{attribute addProperty BoxType "EK1122-0000-0018"}
{attribute addProperty Id "Beckhoff_EP3xxxsub_EK1100EK1100_179A0949162A_0001_EP3162_0002_0016EP3162_C6F348DD14618.25A_0002_EP3162_1002_0017EP3162_F6B2922016220.25A_0003_EP3174_0002_0016EP3174_360D511E40650.75A_0004_EP3174_0002_0017EP3174_360D511E40650.75A_0005_EP3174_0002_0018EP3174_6082EBFD21026.25A_0006_EP3174_0002_0019EP3174_6082EBFD21026.25A_0007_EP3174_0002_0020EP3174_B7B5302521026.25A_0008_EP3174_0002_0021EP3174_B7B5302521026.25A_0009_EP3174_0002_0022EP3174_B7B5302521026.25A_0010_EP3174_0002_0023EP3174_B7B5302521026.25A_0011_EP3174_0092_0016EP3174_B7B5302521026.25A_0012_EP3182_1002_0017EP3182_12747D8E16220.25A_0013_EP3182_1002_0018EP3182_F6B2922016220.25A_0014_EP3182_1002_0019EP3182_F6B2922016220.25A_0015_EP3182_1002_0020EP3182_F6B2922016220.25A_0016_EP3184_0002_0016EP3184_360D511E40650.75A_0017_EP3184_0002_0017EP3184_6082EBFD21026.25A_0018_EP3184_0002_0018EP3184_6082EBFD21026.25A_0019_EP3184_0002_0019EP3184_6082EBFD21026.25A_0020_EP3184_0002_0020EP3184_6082EBFD21026.25A_0021_EP3184_0002_0021EP3184_B7B5302521026.25A_0022_EP3184_0402_0016EP3184_6082EBFD21026.25A_0023_EP3184_0402_0017EP3184_6082EBFD21026.25A_0024_EP3184_0402_0018EP3184_B7B5302521026.25A_0025_EP3184_1002_0016EP3184_360D511E40650.75A_0026_EP3184_1002_0017EP3184_360D511E40650.75A_0027_EP3184_1002_0018EP3184_6082EBFD21026.25A_0028_EP3184_1002_0019EP3184_6082EBFD21026.25A_0029_EP3184_1002_0020EP3184_6082EBFD21026.25A_0030_EP3184_1002_0021EP3184_B7B5302521026.25A_0031_EP3204_0002_0017EP3204_72ABB95437847.25A_0032_EP3204_0002_0018EP3204_72ABB95437847.25A_0033_EP3204_0002_0019EP3204_72ABB95437847.25A_0034_EP3204_0002_0020EP3204_72ABB95437847.25A_0035_EP3204_0002_0021EP3204_C91659E221026.25A_0036_EP3314_0002_0016EP3314_3064F86237847.25A_0037_EP3314_0002_0017EP3314_3064F86237847.25A_0038_EP3314_0002_0018EP3314_1D3C92AC21026.25A_0039_EP3314_0002_0019EP3314_A69716D721026.25A_0040_EP3314_0002_0020EP3314_A69716D721026.25A_0041_EP3314_0002_0021EP3314_A69716D721026.25A_0042_EP3351_2022_0016EP3351_952A9D2322628.25A_0043_EP3356_0022_0016EP3356_AAE78EE214618.25A_0044_EP3356_0022_0017EP3356_AAE78EE214618.25A_0045_EP3356_0022_0022EP3356_AAE78EE214618.25A_0046_EP3632_0001_0016EP3632_A724E07457872.25A_0047_EP3632_0001_0017EP3632_A724E07457872.25A_0048_EP3744_0041_0016EP3744_99A8040A38648.25A_0049_EP3744_0041_0017EP3744_99A8040A38648.25A_0050_EP3744_0041_0018EP3744_99A8040A38648.25A_0051_EP3744_0041_0019EP3744_99A8040A38648.25A_0052_EP3744_0041_0020EP3744_99A8040A38648.25A_0053_EP3744_0041_0021EP3744_99A8040A38648.25A_0054_EP3744_1041_0016EP3744_99A8040A38648.25A_0055_EP3744_1041_0017EP3744_99A8040A38648.25A_0056_EP3744_1041_0018EP3744_99A8040A38648.25A_0057_EP3744_1041_0019EP3744_99A8040A38648.25A_0058_EP3744_1041_0020EP3744_99A8040A38648.25A_0059_EP3744_1041_0021EP3744_99A8040A38648.25A_0060_EP3752_0000_0017EP3752_639ED5F327434.25A_0061_EP3752_0000_0018EP3752_639ED5F327434.25"}
{attribute addProperty CRC "2518642837"}
{attribute addProperty SizeInBites "17310"}
{attribute addProperty SizeInBytes "2163.75"}
TYPE Beckhoff_EP3xxxEK1122_961F7095 EXTENDS EK1122_179A0949 :
STRUCT
	{attribute addProperty Name "Beckhoff_EP3xxxsub_EK1100"}
	Beckhoff_EP3xxxsub_EK1100 : EK1100_179A0949;
	{attribute addProperty Name "A_0001_EP3162_0002_0016"}
	A_0001_EP3162_0002_0016 : EP3162_C6F348DD;
	{attribute addProperty Name "A_0002_EP3162_1002_0017"}
	A_0002_EP3162_1002_0017 : EP3162_F6B29220;
	{attribute addProperty Name "A_0003_EP3174_0002_0016"}
	A_0003_EP3174_0002_0016 : EP3174_360D511E;
	{attribute addProperty Name "A_0004_EP3174_0002_0017"}
	A_0004_EP3174_0002_0017 : EP3174_360D511E;
	{attribute addProperty Name "A_0005_EP3174_0002_0018"}
	A_0005_EP3174_0002_0018 : EP3174_6082EBFD;
	{attribute addProperty Name "A_0006_EP3174_0002_0019"}
	A_0006_EP3174_0002_0019 : EP3174_6082EBFD;
	{attribute addProperty Name "A_0007_EP3174_0002_0020"}
	A_0007_EP3174_0002_0020 : EP3174_B7B53025;
	{attribute addProperty Name "A_0008_EP3174_0002_0021"}
	A_0008_EP3174_0002_0021 : EP3174_B7B53025;
	{attribute addProperty Name "A_0009_EP3174_0002_0022"}
	A_0009_EP3174_0002_0022 : EP3174_B7B53025;
	{attribute addProperty Name "A_0010_EP3174_0002_0023"}
	A_0010_EP3174_0002_0023 : EP3174_B7B53025;
	{attribute addProperty Name "A_0011_EP3174_0092_0016"}
	A_0011_EP3174_0092_0016 : EP3174_B7B53025;
	{attribute addProperty Name "A_0012_EP3182_1002_0017"}
	A_0012_EP3182_1002_0017 : EP3182_12747D8E;
	{attribute addProperty Name "A_0013_EP3182_1002_0018"}
	A_0013_EP3182_1002_0018 : EP3182_F6B29220;
	{attribute addProperty Name "A_0014_EP3182_1002_0019"}
	A_0014_EP3182_1002_0019 : EP3182_F6B29220;
	{attribute addProperty Name "A_0015_EP3182_1002_0020"}
	A_0015_EP3182_1002_0020 : EP3182_F6B29220;
	{attribute addProperty Name "A_0016_EP3184_0002_0016"}
	A_0016_EP3184_0002_0016 : EP3184_360D511E;
	{attribute addProperty Name "A_0017_EP3184_0002_0017"}
	A_0017_EP3184_0002_0017 : EP3184_6082EBFD;
	{attribute addProperty Name "A_0018_EP3184_0002_0018"}
	A_0018_EP3184_0002_0018 : EP3184_6082EBFD;
	{attribute addProperty Name "A_0019_EP3184_0002_0019"}
	A_0019_EP3184_0002_0019 : EP3184_6082EBFD;
	{attribute addProperty Name "A_0020_EP3184_0002_0020"}
	A_0020_EP3184_0002_0020 : EP3184_6082EBFD;
	{attribute addProperty Name "A_0021_EP3184_0002_0021"}
	A_0021_EP3184_0002_0021 : EP3184_B7B53025;
	{attribute addProperty Name "A_0022_EP3184_0402_0016"}
	A_0022_EP3184_0402_0016 : EP3184_6082EBFD;
	{attribute addProperty Name "A_0023_EP3184_0402_0017"}
	A_0023_EP3184_0402_0017 : EP3184_6082EBFD;
	{attribute addProperty Name "A_0024_EP3184_0402_0018"}
	A_0024_EP3184_0402_0018 : EP3184_B7B53025;
	{attribute addProperty Name "A_0025_EP3184_1002_0016"}
	A_0025_EP3184_1002_0016 : EP3184_360D511E;
	{attribute addProperty Name "A_0026_EP3184_1002_0017"}
	A_0026_EP3184_1002_0017 : EP3184_360D511E;
	{attribute addProperty Name "A_0027_EP3184_1002_0018"}
	A_0027_EP3184_1002_0018 : EP3184_6082EBFD;
	{attribute addProperty Name "A_0028_EP3184_1002_0019"}
	A_0028_EP3184_1002_0019 : EP3184_6082EBFD;
	{attribute addProperty Name "A_0029_EP3184_1002_0020"}
	A_0029_EP3184_1002_0020 : EP3184_6082EBFD;
	{attribute addProperty Name "A_0030_EP3184_1002_0021"}
	A_0030_EP3184_1002_0021 : EP3184_B7B53025;
	{attribute addProperty Name "A_0031_EP3204_0002_0017"}
	A_0031_EP3204_0002_0017 : EP3204_72ABB954;
	{attribute addProperty Name "A_0032_EP3204_0002_0018"}
	A_0032_EP3204_0002_0018 : EP3204_72ABB954;
	{attribute addProperty Name "A_0033_EP3204_0002_0019"}
	A_0033_EP3204_0002_0019 : EP3204_72ABB954;
	{attribute addProperty Name "A_0034_EP3204_0002_0020"}
	A_0034_EP3204_0002_0020 : EP3204_72ABB954;
	{attribute addProperty Name "A_0035_EP3204_0002_0021"}
	A_0035_EP3204_0002_0021 : EP3204_C91659E2;
	{attribute addProperty Name "A_0036_EP3314_0002_0016"}
	A_0036_EP3314_0002_0016 : EP3314_3064F862;
	{attribute addProperty Name "A_0037_EP3314_0002_0017"}
	A_0037_EP3314_0002_0017 : EP3314_3064F862;
	{attribute addProperty Name "A_0038_EP3314_0002_0018"}
	A_0038_EP3314_0002_0018 : EP3314_1D3C92AC;
	{attribute addProperty Name "A_0039_EP3314_0002_0019"}
	A_0039_EP3314_0002_0019 : EP3314_A69716D7;
	{attribute addProperty Name "A_0040_EP3314_0002_0020"}
	A_0040_EP3314_0002_0020 : EP3314_A69716D7;
	{attribute addProperty Name "A_0041_EP3314_0002_0021"}
	A_0041_EP3314_0002_0021 : EP3314_A69716D7;
	{attribute addProperty Name "A_0042_EP3351_2022_0016"}
	A_0042_EP3351_2022_0016 : EP3351_952A9D23;
	{attribute addProperty Name "A_0043_EP3356_0022_0016"}
	A_0043_EP3356_0022_0016 : EP3356_AAE78EE2;
	{attribute addProperty Name "A_0044_EP3356_0022_0017"}
	A_0044_EP3356_0022_0017 : EP3356_AAE78EE2;
	{attribute addProperty Name "A_0045_EP3356_0022_0022"}
	A_0045_EP3356_0022_0022 : EP3356_AAE78EE2;
	{attribute addProperty Name "A_0046_EP3632_0001_0016"}
	A_0046_EP3632_0001_0016 : EP3632_A724E074;
	{attribute addProperty Name "A_0047_EP3632_0001_0017"}
	A_0047_EP3632_0001_0017 : EP3632_A724E074;
	{attribute addProperty Name "A_0048_EP3744_0041_0016"}
	A_0048_EP3744_0041_0016 : EP3744_99A8040A;
	{attribute addProperty Name "A_0049_EP3744_0041_0017"}
	A_0049_EP3744_0041_0017 : EP3744_99A8040A;
	{attribute addProperty Name "A_0050_EP3744_0041_0018"}
	A_0050_EP3744_0041_0018 : EP3744_99A8040A;
	{attribute addProperty Name "A_0051_EP3744_0041_0019"}
	A_0051_EP3744_0041_0019 : EP3744_99A8040A;
	{attribute addProperty Name "A_0052_EP3744_0041_0020"}
	A_0052_EP3744_0041_0020 : EP3744_99A8040A;
	{attribute addProperty Name "A_0053_EP3744_0041_0021"}
	A_0053_EP3744_0041_0021 : EP3744_99A8040A;
	{attribute addProperty Name "A_0054_EP3744_1041_0016"}
	A_0054_EP3744_1041_0016 : EP3744_99A8040A;
	{attribute addProperty Name "A_0055_EP3744_1041_0017"}
	A_0055_EP3744_1041_0017 : EP3744_99A8040A;
	{attribute addProperty Name "A_0056_EP3744_1041_0018"}
	A_0056_EP3744_1041_0018 : EP3744_99A8040A;
	{attribute addProperty Name "A_0057_EP3744_1041_0019"}
	A_0057_EP3744_1041_0019 : EP3744_99A8040A;
	{attribute addProperty Name "A_0058_EP3744_1041_0020"}
	A_0058_EP3744_1041_0020 : EP3744_99A8040A;
	{attribute addProperty Name "A_0059_EP3744_1041_0021"}
	A_0059_EP3744_1041_0021 : EP3744_99A8040A;
	{attribute addProperty Name "A_0060_EP3752_0000_0017"}
	A_0060_EP3752_0000_0017 : EP3752_639ED5F3;
	{attribute addProperty Name "A_0061_EP3752_0000_0018"}
	A_0061_EP3752_0000_0018 : EP3752_639ED5F3;
END_STRUCT
END_TYPE

(* stored: Version 1.2.0.0, ProductVersion 3.1.4024.9
   DUT Beckhoff_EP3xxxEK1122_961F7095: Id {861e0a22-2bbe-44f9-a30f-5fed476f6ea7} *)
